FUNCTION TryConvert_LINT_TO_DINT : BOOL
VAR_INPUT
	in : LINT;
	out : REFERENCE TO DINT;
END_VAR

IF in > DatatypeLimits.MAX_VALUE_OF_LINT_WHICH_CAN_BE_HELD_IN_A_DINT THEN
	RETURN;
END_IF

IF in < DatatypeLimits.MIN_VALUE_OF_LINT_WHICH_CAN_BE_HELD_IN_A_DINT THEN
	RETURN;
END_IF

out := LINT_TO_DINT(in);
TryConvert_LINT_TO_DINT := TRUE;

END_FUNCTION

(* stored: Version 1.1.0.1, ProductVersion 3.1.4024.12
   POU TryConvert_LINT_TO_DINT: Id {542ccc19-22f6-4acf-a37f-eb72c0a1e081}, SpecialFunc None *)
